FUNCTION_BLOCK ABSTRACT FB_Actor2Point
VAR_INPUT
	//internal input variables:
	bSetStatusOnAutomatic : BOOL; //turn actor on
	algorithmPermission : BOOL; //is true if control by algorithm is allowed
END_VAR
VAR_OUTPUT
END_VAR
VAR
	//OPC UA structured variables:
	{attribute 'OPC.UA.DA' := '1'}
	control : ST_Control;
	{attribute 'OPC.UA.DA' := '1'}
	controlState : ST_ControlState;
	{attribute 'OPC.UA.DA' := '1'}
	errorState : ST_ErrorState;

	//internal variables:
	bSetStatusOn : BOOL; //actual internal value to switch on 
END_VAR

PROPERTY bStatusOn : BOOL
GET
bStatusOn := controlState.bStatusOn;
END_GET
END_PROPERTY

METHOD PROTECTED SelectControlMode : BOOL
VAR_INPUT
END_VAR

VAR
END_VAR
//change access mode
IF control.bManualModeActivated THEN
	controlState.nAccessmode := E_SystemControlState.manual;
	controlState.sAccessMode := 'manual';
	bSetStatusOn := control.bSetStatusOnManual;
ELSIF control.bAlgorithmModeActivated AND algorithmPermission THEN
	controlState.nAccessmode := E_SystemControlState.algorithm;
	controlState.sAccessMode := 'algorithm';
	bSetStatusOn := control.bSetStatusOnAlgorithm;
ELSE
	controlState.nAccessmode := E_SystemControlState.automatic;
	controlState.sAccessMode := 'automatic';
	bSetStatusOn := bSetStatusOnAutomatic;
END_IF
END_METHOD

END_FUNCTION_BLOCK

(* stored: Version 1.1.0.1, ProductVersion 3.1.4024.9
   POU FB_Actor2Point: Id {779c39b8-c120-47da-8edf-760811555f3b}, SpecialFunc None
   Property bStatusOn: Id {8d0a9f66-53f0-4faa-aec7-56f3439086a4}
   Get Get: Id {996681ce-1125-4289-a2ab-680a8f58a25d}
   Method SelectControlMode: Id {3e578076-f21b-4cb6-b8d9-37cde3c10288} *)
